RoboDK station: Station1.rdk

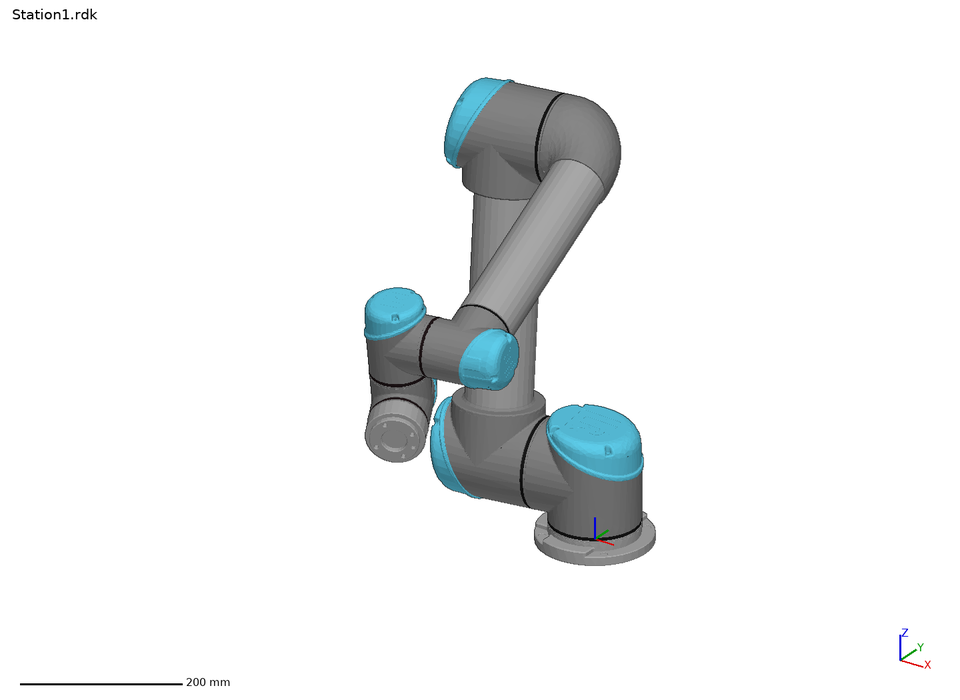
[picture v0: the station drawn from its stored meshes, robots at their saved joint values, targets as dots, program paths as lines]
Station Station1 (saved by RoboDK 5.6.0). Poses are relative to the parent item; angles as X-Y-Z fixed-axis rotations.
  - frame UR5 Base at (0, 0, 0) mm
    - robot UR5: 6 axes
        modified DH rows (alpha deg, a mm, theta deg, d mm): 0, 0, 0, 89.2; 90, 0, 180, 0; 0, 425, 0, 0; 0, 392, 0, 109.3; -90, 0, 0, 94.75; 90, 0, 0, 82.5
        joint limits [-360, -360, -360, -360, -360, -360] to [360, 360, 360, 360, 360, 360]; home [0, -90, -90, 0, 90, 0]; saved at [-81.026, -84.223, -113.165, -172.539, -108.625, 67.737]
  - Python program MoveRobot (listed below)

--- Python program MoveRobot ---
from robolink import Robolink, Item

class MoveRobot:
    def __init__(self):
        self.robodk = Robolink()
        self.station = self.robodk.AddFile('Station1.rdk')


    def move_robot_to_point(self, point):
        pass  # Implement the movement logic here
